TYPE SC_SENSOR_BeltConveyors :
(
	eCounterSensor := 1,
	eBeltConveyorsMaxSensors
)UINT;
END_TYPE

(* stored: Version 1.1.0.1, ProductVersion 3.1.4024.0
   DUT SC_SENSOR_BeltConveyors: Id {fba731ae-a66e-47a4-9c19-af5c6ec300dd} *)
